{attribute 'GeneratedUsingTerminal: EL5101-0011-0016'}
{attribute addProperty BoxType "EL5101-0011-0016"}
{attribute addProperty Id "Counter_valueAT %I*Counter_value_E1FCE22B4"}
{attribute addProperty CRC "559421638"}
{attribute addProperty Size "4"}
TYPE ENC_TxPdo_1_Samples_Counter_value_215818C6 :
STRUCT
	{attribute addProperty Name "Counter_value"}
	Counter_value AT %I* : Counter_value_E1FCE22B;
END_STRUCT
END_TYPE

(* stored: Version 1.2.0.0, ProductVersion 3.1.4024.9
   DUT ENC_TxPdo_1_Samples_Counter_value_215818C6: Id {fa82b7ac-0636-4381-ac3f-d4405505e8b1} *)
